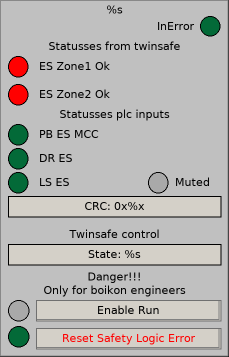
VISUALIZATION Vis_SafetyZone1  // 229x357
VAR_INPUT
	I_Title:string;
END_VAR

VAR_IN_OUT
	IO_SafetyLogic:cntrl_SafetyController1;
END_VAR
    Rectangle (0,0 229x357)
    Rectangle (12,0 205x20), "%s", text variable: I_Title
    Rectangle (8,244 213x21), "State: %s", text variable: IO_SafetyLogic.eS
    Button (36,328 185x21), "Reset Safety Logic Error", pressed state: IO_SafetyLogic.PbSf_ResetSafetyErrors.P_BypassStateTrue
        tap IO_SafetyLogic.PbSf_ResetSafetyErrors.P_BypassStateTrue
    Ellipse (8,326 21x21), colour toggle: IO_SafetyLogic.HMI.STS.LogicInError
    Ellipse (8,300 21x21), colour toggle: IO_SafetyLogic.HMI.STS.LogicRunning
    Rectangle (8,268 213x31), "Danger!!! Only for boikon engineers"
    Button (36,300 185x21), "Enable Run", pressed state: IO_SafetyLogic.HMI.STS.PB_RunSafetyLogic
        toggle IO_SafetyLogic.HMI.STS.PB_RunSafetyLogic
    Ellipse (8,56 20x21), colour toggle: IO_SafetyLogic.Isf_STS_ES_Zone1_OK.HMI.STS.State
    Rectangle (36,56 181x21), "ES Zone1 Ok"
    Ellipse (8,124 20x21), colour toggle: NOT IO_SafetyLogic.PB_ES_MainCabinet.HMI.STS.StateOk
    Rectangle (36,124 181x21), "PB ES MCC"
    Ellipse (8,148 20x21), colour toggle: NOT IO_SafetyLogic.DR_Front.HMI.STS.StateOk
    Rectangle (36,148 181x21), "DR ES"
    Ellipse (8,172 20x21), colour toggle: NOT IO_SafetyLogic.LS_Entry1.HMI.STS.StateOk
    Rectangle (36,172 73x21), "LS ES"
    Ellipse (200,16 20x20), colour toggle: IO_SafetyLogic.HMI.P_STS_InError
    Rectangle (128,16 69x21), "InError"
    Label (8,36 213x21), "Statusses from twinsafe"
    Label (8,104 213x21), "Statusses plc inputs"
    Label (8,224 213x21), "Twinsafe control"
    Rectangle (8,196 213x21), "CRC: 0x%x", text variable: IO_SafetyLogic.HMI.STS.CrcCodeProject
    Ellipse (8,84 20x21), colour toggle: IO_SafetyLogic.Isf_STS_ES_Zone2_OK.HMI.STS.State
    Rectangle (36,84 181x21), "ES Zone2 Ok"
    Ellipse (148,172 20x21), colour toggle: IO_SafetyLogic.LS_Entry1.HMI.STS.StateMuted
    Rectangle (172,172 49x21), "Muted"
END_VISUALIZATION

(* stored: Version 1.1.0.1
   Visu Vis_SafetyZone1: Id {5a4749fc-7e5d-02c1-105b-1be2175978d8} *)
